FUNCTION_BLOCK Axis_Power
VAR_INPUT
	SpeedControl:INT;
END_VAR
VAR_OUTPUT
	Power_Status:BOOL;
END_VAR
VAR
	AxisPower1: MC_Power;
	AxisPower2: MC_Power;
END_VAR

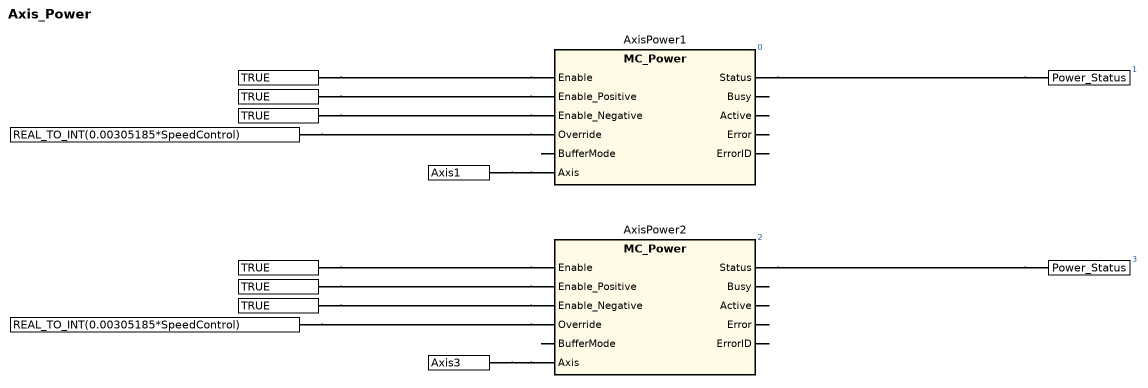
AxisPower1(
    Enable := TRUE,
    Enable_Positive := TRUE,
    Enable_Negative := TRUE,
    Override := REAL_TO_INT(0.00305185*SpeedControl),
    Axis := Axis1); // MC_Power
Power_Status := AxisPower1.Status;
AxisPower2(
    Enable := TRUE,
    Enable_Positive := TRUE,
    Enable_Negative := TRUE,
    Override := REAL_TO_INT(0.00305185*SpeedControl),
    Axis := Axis3); // MC_Power
Power_Status := AxisPower2.Status;

END_FUNCTION_BLOCK

(* stored: Version 1.1.0.1, ProductVersion 3.1.4024.12
   POU Axis_Power: Id {888f4209-dbae-495c-bfe7-6f9198cdea21}, SpecialFunc None *)
